// TIA Portal V15.1 export
// export: Created 2026-01-09T13:45:13.0471947Z, ExportSetting WithDefaults, WithReadOnly, DisplayName Totally Integrated Automation Portal, DisplayVersion V15.1 Update 8, DisplayName TIA Portal Openness, DisplayVersion V15.1 Update 8, DisplayName STEP 7 Professional, DisplayVersion V15.1 Update 8, DisplayName WinCC Advanced, DisplayVersion V15.1 Update 8
DATA_BLOCK "2.0_NN0_0"   // DB200
{ S7_Optimized_Access := 'TRUE' }
VERSION : 0.1
// stored: AutoNumber false, CodeModifiedDate 2025-08-27T17:14:33.7093845Z, CompileDate 2025-08-30T17:40:34.5623931Z, CreationDate 2024-10-12T12:36:08.0193576Z, DBAccessibleFromOPCUA true, DownloadWithoutReinit false, InstanceOfName 2.MANUAL_CONTROL, InstanceOfNumber 2, InstanceOfType FB, InterfaceModifiedDate 2025-08-27T17:14:33.2091456Z, IsConsistent true, IsKnowHowProtected false, IsRetainMemResEnabled false, MemoryReserve 100, ModifiedDate 2025-08-27T17:14:33.7093845Z, ParameterModified 2024-10-13T14:59:19.5830719Z, StructureModified 2025-08-27T17:14:33.2091456Z, UDAEnableTagReadback false
"2.MANUAL_CONTROL"
   // VAR_INPUT
   //    MODE : Bool;
   //    NN1 : Bool;
   //    NN2 : Bool;
   //    NN3 : Bool;
   //    ST1 : Bool;
   //    ST2 : Bool;
   //    ST3 : Bool;
   //    RS1 : Bool;
   //    RS2 : Bool;
   //    RS3 : Bool;
   // END_VAR
   // VAR_OUTPUT
   //    OUT1 : Bool;
   //    OUT2 : Bool;
   //    OUT3 : Bool;
   // END_VAR
   // VAR
   //    OUT11 : Bool;
   //    OUT12 : Bool;
   //    OUT21 : Bool;
   //    OUT22 : Bool;
   //    OUT31 : Bool;
   //    OUT32 : Bool;
   //    M1 : Int;
   //    M2 : Int;
   //    M3 : Int;
   //    M4 : Bool;
   //    M5 : Bool;
   //    M6 : Bool;
   // END_VAR
BEGIN
END_DATA_BLOCK
